      # find rxryrz1
      # first rotation is 135 degrees about the y- direction. 90 degrees to get flat. Tip pointing x-, preheat pointing y+. 45 more degrees to get at that above angle
      m1 = get_rotation_matrix_from_description("y", -1, 135 * pi / 180)
      # second rotation is heading1 – 180 degrees about the z+ axis to get pointing straight into wall. Heading1 should be about 180 degrees
      m2 = get_rotation_matrix_from_description("z", 1, heading1 - 180 * pi/180)
      # combine them by multiplying
      m3 = multiply_matrix(m2, m1)
      rxryrz1 = convert_matrix_to_axang(m3)
      rx1 = rxryrz1[0]
      ry1 = rxryrz1[1]
      rz1 = rxryrz1[2]

      point1 = p[p1x, p1y, p1z, rx1, ry1, rz1]

      # get second point (right) (point2)
      # take the center point and move right the radius plus the cushions
      p2x = pcx + vecrx * radius + vecrx * cusharound + vecnx * -1 * cushout
      p2y = pcy + vecry * radius + vecry * cusharound + vecny * -1 * cushout
      p2z = pcz

      # find rxryrz2
      # first rotation is 90 degrees about the x- axis
      m1 = get_rotation_matrix_from_description("x", -1, 90 * pi / 180)
      # second rotation is About 135 degrees about the z+ axis. This calculation is heading1 – 45 degrees
      m2 = get_rotation_matrix_from_description("z", 1, heading1 - 45 * pi/180)
      # combine them by multiplying
      m3 = multiply_matrix(m2, m1)
      rxryrz2 = convert_matrix_to_axang(m3)
      rx2 = rxryrz2[0]
      ry2 = rxryrz2[1]
      rz2 = rxryrz2[2]

      point2 = p[p2x, p2y, p2z, rx2, ry2, rz2]

      # get the third point (bottom) (point3)
      p3x = pcx + vecnx * -1 * cushout
      p3y = pcy + vecny * -1 * cushout
      p3z = pcz - vecuz * radius - vecuz * cusharound

      # find rxryrz3
      # first rotation is 45 degrees about the y+ axis
      m1 = get_rotation_matrix_from_description("y", 1, 45 * pi / 180)
      # second rotation is About 180 degrees about the z+ axis. This calculation is heading1 degrees
      m2 = get_rotation_matrix_from_description("z", 1, heading1)
      # combine them by multiplying
      m3 = multiply_matrix(m2, m1)
      rxryrz3 = convert_matrix_to_axang(m3)
      rx3 = rxryrz3[0]
      ry3 = rxryrz3[1]
      rz3 = rxryrz3[2]

      point3 = p[p3x, p3y, p3z, rx3, ry3, rz3]

      # get the fourth point (left) (point4)
      p4x = pcx - vecrx * radius - vecrx * cusharound + vecnx * -1 * cushout
      p4y = pcy - vecry * radius - vecry * cusharound + vecny * -1 * cushout
      p4z = pcz

      # find rxryrz4
      # first rotation is 90 degrees about the x+ axis
      m1 = get_rotation_matrix_from_description("x", 1, 90 * pi / 180)
      # second rotation is heading1 + 45 degrees about the z+ axis. approx 225 degrees ccw
      m2 = get_rotation_matrix_from_description("z", 1, heading1 + 45 * pi/180)
      # combine them by multiplying
      m3 = multiply_matrix(m2, m1)
      rxryrz4 = convert_matrix_to_axang(m3)
      rx4 = rxryrz4[0]
      ry4 = rxryrz4[1]
      rz4 = rxryrz4[2]

      point4 = p[p4x, p4y, p4z, rx4, ry4, rz4]

      # get the angle for the tilt-back at the top (p1)
      m0 = get_rotation_matrix_from_description("x", -1, 10 * pi / 180)
      m1 = get_rotation_matrix_from_description("y", -1, 135 * pi / 180)
      # second rotation is heading1 – 180 degrees about the z+ axis to get pointing straight into wall. Heading1 should be about 180 degrees
      m2 = get_rotation_matrix_from_description("z", 1, heading1 - 180 * pi/180)
      # combine them by multiplying
      m3 = multiply_matrix(m2, m1)
      m4 = multiply_matrix(m3, m0)
      rxryrz1tilt = convert_matrix_to_axang(m4)
      rx1t = rxryrz1tilt[0]
      ry1t = rxryrz1tilt[1]
      rz1t = rxryrz1tilt[2]

      # point 1, but with the tilt back angle
      point1t = p[p1x, p1y, p1z, rx1t, ry1t, rz1t]

      # point45 (the point 45 degrees along the path) (has no rxryrz data) (because if we do fixed angle circle move it wont use that anyways, it'l just use the angle from p1t)
      distup = cos(45 * pi/180) * (radius + cusharound)
      distover = sin(45 * pi/180) * (radius + cusharound)
      p45x = pcx + vecrx * distover + vecnx * -1 * cushout
      p45y = pcy + vecry * distover + vecny * -1 * cushout
      p45z = pcz + vecuz * distup
      point45 = p[p45x, p45y, p45z, 0,0,0]

      # point22 (22.5 degrees of angle)
      distup = cos(22.5 * pi/180) * (radius + cusharound)
      distover = sin(22.5 * pi/180) * (radius + cusharound)
      p22x = pcx + vecrx * distover + vecnx * -1 * cushout
      p22y = pcy + vecry * distover + vecny * -1 * cushout
      p22z = pcz + vecuz * distup
      point22 = p[p22x, p22y, p22z, 0,0,0]

      # return the points
      ret = struct(point1=point1, point2=point2, point3=point3, point4=point4, point1t=point1t, point45=point45, point22=point22)
      return ret

  end

  def make_pose_list(length):
      if length < 1:
          ret = []
          return ret
      end
      if length == 1:
          pose_list = [p[0, 0, 0, 0, 0, 0]]
          return pose_list
      end
      if length == 2:
          pose_list = [p[0, 0, 0, 0, 0, 0], p[0, 0, 0, 0, 0, 0]]
          return pose_list
      end
      if length == 3:
          pose_list = [p[0, 0, 0, 0, 0, 0], p[0, 0, 0, 0, 0, 0], p[0, 0, 0, 0, 0, 0]]
          return pose_list
      end
      if length == 4:
          pose_list = [p[0, 0, 0, 0, 0, 0], p[0, 0, 0, 0, 0, 0], p[0, 0, 0, 0, 0, 0], p[0, 0, 0, 0, 0, 0]]
          return pose_list
      end
      if length == 5:
          pose_list = [p[0, 0, 0, 0, 0, 0], p[0, 0, 0, 0, 0, 0], p[0, 0, 0, 0, 0, 0], p[0, 0, 0, 0, 0, 0], p[0, 0, 0, 0, 0, 0]]
          return pose_list
      end
      if length == 6:
          pose_list = [p[0, 0, 0, 0, 0, 0], p[0, 0, 0, 0, 0, 0], p[0, 0, 0, 0, 0, 0], p[0, 0, 0, 0, 0, 0], p[0, 0, 0, 0, 0, 0], p[0, 0, 0, 0, 0, 0]]
          return pose_list
      end
      if length == 7:
          pose_list = [p[0, 0, 0, 0, 0, 0], p[0, 0, 0, 0, 0, 0], p[0, 0, 0, 0, 0, 0], p[0, 0, 0, 0, 0, 0], p[0, 0, 0, 0, 0, 0], p[0, 0, 0, 0, 0, 0], p[0, 0, 0, 0, 0, 0]]
          return pose_list
      end
      if length == 8:
          pose_list = [p[0, 0, 0, 0, 0, 0], p[0, 0, 0, 0, 0, 0], p[0, 0, 0, 0, 0, 0], p[0, 0, 0, 0, 0, 0], p[0, 0, 0, 0, 0, 0], p[0, 0, 0, 0, 0, 0], p[0, 0, 0, 0, 0, 0], p[0, 0, 0, 0, 0, 0]]
          return pose_list
      end
      if length == 9:
          pose_list = [p[0, 0, 0, 0, 0, 0], p[0, 0, 0, 0, 0, 0], p[0, 0, 0, 0, 0, 0], p[0, 0, 0, 0, 0, 0], p[0, 0, 0, 0, 0, 0], p[0, 0, 0, 0, 0, 0], p[0, 0, 0, 0, 0, 0], p[0, 0, 0, 0, 0, 0], p[0, 0, 0, 0, 0, 0]]
          return pose_list
      end
      if length > 9:
          popuptext = "Program is only capable of storing 9 pegs at once. You selected more than 9. "
          # infinite loop
          while 1==1:
              popup(popuptext, title="Too Many Pegs",blocking=True)
          end
      end
  end

  # this function calculates the poses required on the weldpath for a specific teach pose for peg center.
  # call this function for every peg you want to weld.
  def main_calculate_peg(pose1):
      # constants
      peg_width = 2.05 # inches
      fixture_height = 1.5 # inches
      cushout = 0.006 # 5mm # the cushion out from the wall
      cusharound = 0.004 # 5mm # the cushion around the sleeve.
      delz = fixture_height *25.4/1000 - cushout
      rad = peg_width *1/2 * 25.4/1000 + cusharound

      # calculate angles
      # rxryrz1 (for point 1 (back side of peg)
      # start with gun facing up, shield tip pointing in x+ direction
      # rotate about y axis (y-) 135 degrees.
      # thats it. (for the other ones, then rotate 90 degrees about z axis from this spot
      m0 = get_rotation_matrix_from_description("y", -1, 225 * pi / 180)
      rxryrz1 = convert_matrix_to_axang(m0)
      rx1 = rxryrz1[0]
      ry1 = rxryrz1[1]
      rz1 = rxryrz1[2]

      # rxryrz2
      # second rotation is 90 degrees about z- axis
      m1 = get_rotation_matrix_from_description("z", -1, 90 * pi / 180)
      m2 = multiply_matrix(m1, m0)
      rxryrz2 = convert_matrix_to_axang(m2)
      rx2 = rxryrz2[0]
      ry2 = rxryrz2[1]
      rz2 = rxryrz2[2]

      # rxryrz3
      # second rotation is 180 degrees about z- axis
      m1 = get_rotation_matrix_from_description("z", -1, 180 * pi / 180)
      m2 = multiply_matrix(m1, m0)
      rxryrz3 = convert_matrix_to_axang(m2)
      rx3 = rxryrz3[0]
      ry3 = rxryrz3[1]
      rz3 = rxryrz3[2]

      # rxryrz4
      # second rotation is 270 degrees about z- axis
      m1 = get_rotation_matrix_from_description("z", -1, 270 * pi / 180)
      m2 = multiply_matrix(m1, m0)
      rxryrz4 = convert_matrix_to_axang(m2)
      rx4 = rxryrz4[0]
      ry4 = rxryrz4[1]
      rz4 = rxryrz4[2]

      # get points
      # get lift column height based on z value
      # if z is between +1 feet and -1 feet then go to 750
      # if z is greater than +1 feet but less than +4 feet, then go to 880
      # if z is greater than +4 feet, then error
      # if z is less than -1 feet, then go to 750 mm above z.

      # scrap that. new rules
      # go to 750 mm above z.
      # if that result is above 880, then go to 880.
      # that will work until we get problems

      z0 = pose1[2] # the teach point's z value (taken when lift column = 0)
      lczn = z0 + .750 # lift column z needed
      if lczn > .880:
          lczn = .880
      end
      liftcolumnzneeded = lczn * 1000 # set the z position
      zposerel = z0 - lczn # z pose relative = the teach point's z value at the new lift column position.

      pcenterx = pose1[0]
      pcentery = pose1[1]

      #points
      p1x = pcenterx - rad
      p1y = pcentery
      p1z = zposerel - delz

      p2x = pcenterx
      p2y = pcentery + rad
      p2z = zposerel - delz

      p3x = pcenterx + rad
      p3y = pcentery
      p3z = zposerel - delz

      p4x = pcenterx
      p4y = pcentery - rad
      p4z = zposerel - delz

      point1 = p[p1x, p1y, p1z, rx1, ry1, rz1]
      point2 = p[p2x, p2y, p2z, rx2, ry2, rz2]
      point3 = p[p3x, p3y, p3z, rx3, ry3, rz3]
      point4 = p[p4x, p4y, p4z, rx4, ry4, rz4]

      ret = struct(point1=point1, point2=point2, point3=point3, point4=point4, liftcolumnzneeded=liftcolumnzneeded)
      return ret



  end
  $ 98 "sidewallchoice≔'Is the floor 3/4 inch?'"
  global sidewallchoice=request_boolean_from_primary_client("Is the floor 3/4 inch?")
  $ 99 "If sidewallchoice"
  if (sidewallchoice):
    $ 100 "sidewall≔0.628"
    global sidewall=0.628
  else:
    $ 101 "Else" "noBreak"
    $ 102 "sidewall≔0.375"
    global sidewall=0.375
  end
  $ 106 "Set"
  set_tcp(p[-0.00549,-0.328,0.10639,1.2092,-1.2092,1.2092])
  $ 107 "MoveJ"
  $ 108 "Waypoint_75" "breakAfter"
  movej(get_inverse_kin(Waypoint_75_p, qnear=Waypoint_75_q), a=1.3962634015954636, v=1.0471975511965976)
  $ 109 "Set"
  set_tcp(p[0.0027,-0.0049299999999999995,0.2846,0.0,0.0,0.0])
  $ 110 "MoveJ"
  $ 112 "Waypoint_21" "breakAfter"
  movej(get_inverse_kin(Waypoint_21_p, qnear=Waypoint_21_q), a=1.3962634015954636, v=1.0471975511965976)
  $ 113 "Test_Teach_Straight()"
  Test_Teach_Straight()
  $ 114 "Set"
  set_tcp(p[0.0027,-0.0049299999999999995,0.2846,0.0,0.0,0.0])
  $ 115 "kill threadId_Thread_1"
  kill threadId_Thread_1
  $ 116 "Straight_Homing_Floor_2()"
  Straight_Homing_Floor_2()
  $ 117 "Set"
  set_tcp(p[-0.00549,-0.328,0.10639,1.2092,-1.2092,1.2092])
  $ 122 "pathturn≔main_calculate_floor_straight(p11,p12,p21,p22,sidewall, tcp_pose_left, tcp_pose_right)"
  global pathturn=main_calculate_floor_straight(p11,p12,p21,p22,sidewall, tcp_pose_left, tcp_pose_right)
  $ 123 "extrude_knife3()"
  extrude_knife3()
  $ 129 "align_for_floor_straight()"
  align_for_floor_straight()
  $ 130 "move_path_floor_straight()"
  move_path_floor_straight()
  $ 135 "Home"
  movej([-3.266929759358355, -1.2139462677784536, 1.5878387874396154, 1.1069165929565088, -0.0023738326664366483, -1.7891447305770605], a=1.3962634015954636, v=1.0471975511965976)
end
